# EPICS substitutions: kstar/siteApp/TS1/TS1App/Db/ts_mean_B2.substitutions
#
file db/TS_CH_value.db
{
    pattern
        { DEV,    ID,       TAIL,     DESC,                ARG     }

        {"B2",    "0",      "MEAN",   "mean value",    "raw_mean"}
        {"B2",    "1",       "MEAN",   "mean value",    "raw_mean"}
        {"B2",    "2",       "MEAN",   "mean value",    "raw_mean"}
        {"B2",    "3",       "MEAN",   "mean value",    "raw_mean"}
        {"B2",    "4",       "MEAN",   "mean value",    "raw_mean"}
        {"B2",    "5",       "MEAN",   "mean value",    "raw_mean"}
        {"B2",    "6",       "MEAN",   "mean value",    "raw_mean"}
        {"B2",    "7",       "MEAN",   "mean value",    "raw_mean"}
        {"B2",    "8",       "MEAN",   "mean value",    "raw_mean"}
        {"B2",    "9",       "MEAN",   "mean value",    "raw_mean"}
        {"B2",    "10",       "MEAN",   "mean value",    "raw_mean"}
        {"B2",    "11",       "MEAN",   "mean value",    "raw_mean"}
        {"B2",    "12",       "MEAN",   "mean value",    "raw_mean"}
        {"B2",    "13",       "MEAN",   "mean value",    "raw_mean"}
        {"B2",    "14",       "MEAN",   "mean value",    "raw_mean"}
        {"B2",    "15",       "MEAN",   "mean value",    "raw_mean"}
        {"B2",    "16",       "MEAN",   "mean value",    "raw_mean"}
        {"B2",    "17",       "MEAN",   "mean value",    "raw_mean"}
        {"B2",    "18",       "MEAN",   "mean value",    "raw_mean"}
        {"B2",    "19",       "MEAN",   "mean value",    "raw_mean"}
        {"B2",    "20",       "MEAN",   "mean value",    "raw_mean"}
        {"B2",    "21",       "MEAN",   "mean value",    "raw_mean"}
        {"B2",    "22",       "MEAN",   "mean value",    "raw_mean"}
        {"B2",    "23",       "MEAN",   "mean value",    "raw_mean"}
        {"B2",    "24",       "MEAN",   "mean value",    "raw_mean"}
        {"B2",    "25",       "MEAN",   "mean value",    "raw_mean"}
        {"B2",    "26",       "MEAN",   "mean value",    "raw_mean"}
        {"B2",    "27",       "MEAN",   "mean value",    "raw_mean"}
        {"B2",    "28",       "MEAN",   "mean value",    "raw_mean"}
        {"B2",    "29",       "MEAN",   "mean value",    "raw_mean"}
        {"B2",    "30",       "MEAN",   "mean value",    "raw_mean"}
        {"B2",    "31",       "MEAN",   "mean value",    "raw_mean"}
#
#
        {"B2",    "0",      "BG_MEAN",   "background mean value",    "bg_mean"}
        {"B2",    "1",      "BG_MEAN",   "background mean value",    "bg_mean"}
        {"B2",    "2",      "BG_MEAN",   "background mean value",    "bg_mean"}
        {"B2",    "3",      "BG_MEAN",   "background mean value",    "bg_mean"}
        {"B2",    "4",      "BG_MEAN",   "background mean value",    "bg_mean"}
        {"B2",    "5",      "BG_MEAN",   "background mean value",    "bg_mean"}
        {"B2",    "6",      "BG_MEAN",   "background mean value",    "bg_mean"}
        {"B2",    "7",      "BG_MEAN",   "background mean value",    "bg_mean"}
        {"B2",    "8",      "BG_MEAN",   "background mean value",    "bg_mean"}
        {"B2",    "9",      "BG_MEAN",   "background mean value",    "bg_mean"}
        {"B2",    "10",      "BG_MEAN",   "background mean value",    "bg_mean"}
        {"B2",    "11",      "BG_MEAN",   "background mean value",    "bg_mean"}
        {"B2",    "12",      "BG_MEAN",   "background mean value",    "bg_mean"}
        {"B2",    "13",      "BG_MEAN",   "background mean value",    "bg_mean"}
        {"B2",    "14",      "BG_MEAN",   "background mean value",    "bg_mean"}
        {"B2",    "15",      "BG_MEAN",   "background mean value",    "bg_mean"}
        {"B2",    "16",      "BG_MEAN",   "background mean value",    "bg_mean"}
        {"B2",    "17",      "BG_MEAN",   "background mean value",    "bg_mean"}
        {"B2",    "18",      "BG_MEAN",   "background mean value",    "bg_mean"}
        {"B2",    "19",      "BG_MEAN",   "background mean value",    "bg_mean"}
        {"B2",    "20",      "BG_MEAN",   "background mean value",    "bg_mean"}
        {"B2",    "21",      "BG_MEAN",   "background mean value",    "bg_mean"}
        {"B2",    "22",      "BG_MEAN",   "background mean value",    "bg_mean"}
        {"B2",    "23",      "BG_MEAN",   "background mean value",    "bg_mean"}
        {"B2",    "24",      "BG_MEAN",   "background mean value",    "bg_mean"}
        {"B2",    "25",      "BG_MEAN",   "background mean value",    "bg_mean"}
        {"B2",    "26",      "BG_MEAN",   "background mean value",    "bg_mean"}
        {"B2",    "27",      "BG_MEAN",   "background mean value",    "bg_mean"}
        {"B2",    "28",      "BG_MEAN",   "background mean value",    "bg_mean"}
        {"B2",    "29",      "BG_MEAN",   "background mean value",    "bg_mean"}
        {"B2",    "30",      "BG_MEAN",   "background mean value",    "bg_mean"}
        {"B2",    "31",      "BG_MEAN",   "background mean value",    "bg_mean"}

}
